INTERFACE I_Brake

PROPERTY BrakeMode : E_StageBrakeMode
GET
END_GET
SET
END_SET
END_PROPERTY

PROPERTY BrakeRelease : BOOL
GET
END_GET
SET
END_SET
END_PROPERTY

PROPERTY MotionState : MC_AxisStates
GET
END_GET
SET
END_SET
END_PROPERTY

END_INTERFACE

(* stored: Version 1.1.0.1
   Itf I_Brake: Id {190f63fb-756a-4791-8091-567b83a9d052}
   Property BrakeMode: Id {0e1c15ff-4c0a-4d96-9240-b1fe98efccae}
   Get Get: Id {b15cfe78-2d78-4dcd-917c-25c11507600e}
   Set Set: Id {5bf7a3f4-b227-41be-a6cc-f465ecf3784b}
   Property BrakeRelease: Id {f7411daa-c129-4ae6-a363-2bb5ae6bae27}
   Get Get: Id {d25d5972-d184-4b87-bbef-d0f446a0a92a}
   Set Set: Id {2536a6a9-3571-4972-98d2-90b38510ce0d}
   Property MotionState: Id {cafc07a5-b9fb-4ac1-ba22-5d5dfe1f79d1}
   Get Get: Id {78bb5d85-d490-4014-9418-45338b45e88d}
   Set Set: Id {bcda3488-774d-4d84-a2e1-b59faaa350a4} *)
